{library PUBLIC}
(* Use this function to open an communication link to a specific device defined by Instance.
A communication link is always opened for read/write.
Return value is true if open was ok otherwise false. *)
FUNCTION DeviceOpen : BOOL
VAR_INPUT
	Instance: 				INT;		(* Instance is an address, use the function ToAddress() to convert station and device number to a valid address. *)
END_VAR

DeviceOpen:=FALSE;
IF _GetInstance(Instance)=INSTANCE_STATUS.INSTANCE_STATUS_FREE THEN
	IF _CheckInstance(Instance) THEN
		IF _AllocateInstance(Instance) THEN
			DeviceOpen:=TRUE;
		END_IF;
	END_IF;
END_IF;

END_FUNCTION

(* stored: Version 1.1.0.1, ProductVersion 3.1.4024.2
   POU DeviceOpen: Id {f3da60b0-2d3a-4666-acd7-e3ed66767f11}, SpecialFunc None *)
